// TIA Portal V18 export
DATA_BLOCK "MB_SERVER_DB"   // DB1
// stored: AutoNumber true, DBAccessibleFromOPCUA true, InstanceOfName MB_SERVER, OfSystemLibElement MB_SERVER, OfSystemLibVersion 5.3
"MB_SERVER"
   // VAR_INPUT
   //    DISCONNECT { ExternalVisible := 'False'} : Bool;
   // END_VAR
   // VAR_OUTPUT
   //    NDR { ExternalVisible := 'False'} : Bool;
   //    DR { ExternalVisible := 'False'} : Bool;
   //    ERROR { ExternalVisible := 'False'} : Bool;
   //    STATUS { ExternalVisible := 'False'} : Word;
   // END_VAR
   // VAR_IN_OUT
   //    MB_HOLD_REG : Variant;
   //    CONNECT : Variant;
   // END_VAR
   // VAR
   //    TCON { S7_SetPoint := 'True'} : TCON;
   //    TSEND { S7_SetPoint := 'True'} : TSEND;
   //    TRCV { S7_SetPoint := 'True'} : TRCV;
   //    TDIAG { S7_SetPoint := 'True'} : T_DIAG;
   //    TRESET { S7_SetPoint := 'True'} : T_RESET;
   //    TDISCON { S7_SetPoint := 'True'} : TDISCON;
   //    TDIAG_Status { S7_SetPoint := 'True'} : TDiag_Status;
   //    HR_Start_Offset : Word;
   //    QB_Start : UInt;
   //    QB_Count : UInt;
   //    QB_Read_Start : UInt;
   //    QB_Read_Count : UInt;
   //    IB_Read_Start : UInt;
   //    IB_Read_Count : UInt;
   //    Success_Count : Word;
   //    Request_Count : Word;
   //    Xmt_Rcv_Count : Word;
   //    Server_Message_Count : Word;
   //    Exception_Count : Word;
   //    Connected : Bool;
   //    Connection_ID { ExternalVisible := 'False'} : Word;
   //    MB_State : Word;
   //    TEMP_DATA { ExternalVisible := 'False'} : Array[0..262] of Byte;
   //    Data_Area_Array { S7_SetPoint := 'True'} : Array[1..8] of MB_DataArea;
   //    NDR_immediate : Bool;
   //    DR_immediate : Bool;
   //    BytesReceived : UDInt;
   //    overflow_buffer : Array[0..262] of Byte;
   //    overflow_size_bytes : UInt;
   // END_VAR
BEGIN
END_DATA_BLOCK
